Universal Robots URScript: pendant_pick_place.urscript

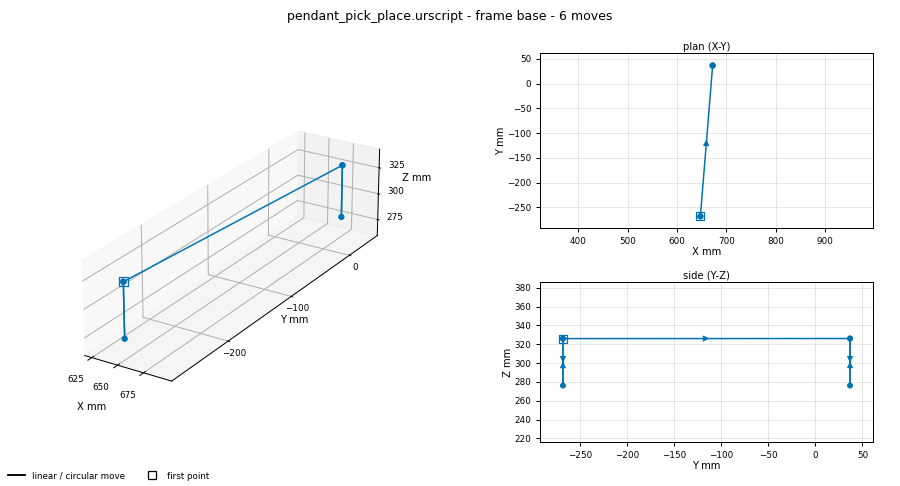
[picture p0: tool path of pendant_pick_place.urscript in frame base, 6 of 6 moves have a stored position in this frame; points joined in program order, loops and branches not executed]
# ===== Robotiq 2F-85 抓取-放置程序（示教器 Script 节点用）=====
# 抓取点: [0.6474,-0.2685,0.2761]  放置点: [0.6722,0.0368,0.2761]

rq_activate()
sleep(0.5)
movel(p[0.6474272729282422,-0.268465964721239,0.32605580637812587,1.9351373451718241,-2.3646005215619694,-0.00022114968079682207], a=0.3, v=0.05)
movel(p[0.6474272729282422,-0.268465964721239,0.2760558063781259,1.9351373451718241,-2.3646005215619694,-0.00022114968079682207], a=0.3, v=0.05)
sleep(0.3)
rq_move_to(255)      # 闭合夹爪
sleep(0.8)
movel(p[0.6474272729282422,-0.268465964721239,0.32605580637812587,1.9351373451718241,-2.3646005215619694,-0.00022114968079682207], a=0.3, v=0.05)
movel(p[0.672239834897491,0.03678128214703258,0.3261125259113394,1.9351373451718241,-2.3646005215619694,-0.00022114968079682207], a=0.3, v=0.05)
movel(p[0.672239834897491,0.03678128214703258,0.2761125259113394,1.9351901513169982,-2.3646862311110817,-2.300586535676707e-05], a=0.3, v=0.05)
sleep(0.3)
rq_move_to(0)        # 张开夹爪
sleep(0.8)
movel(p[0.672239834897491,0.03678128214703258,0.3261125259113394,1.9351373451718241,-2.3646005215619694,-0.00022114968079682207], a=0.3, v=0.05)

# 想循环就取消下面注释（把上面动作包进 while True）
